Universal Robots PolyScope program: urcadpts_urp_ex.urp

Program urcadpts_urp_ex (installation=default directory=/programs createdIn=5.21.0 lastSavedIn=5.21.0 robotSerialNumber=20205500771)
Calibrated DH parameters: a=[0.00017, -0.315777, -0.390584, 0.000089, 0.000022, 0]; d=[0.16289, -151.810109, 155.986099, -4.043122, 0.099816, 0.099706]; alpha=[1.572969, -0.001875, 0.009547, 1.571313, -1.570827, 0]; deltaTheta=[0, 0.733614, -0.631905, -0.101721, 0.000001, 0]
InitVariablesNode
Robot Program (runOnlyOnce=false)
  Folder Folder
    Folder BeforeStart setup urcadpts: load source file, set PCS and orientation
      'use a script node to load the .script file here'
      Script: urcadpts_set_pcs()
      Script: urcadpts_use_pcs_as_orientation( True )
    Folder RobotProgram Example Usage
      Loop While (checkContinuously=false) expression=urcadpts_pts_remaining()≟ True
        target_point := urcadpts_get_next_point()
        approach_point := pose_trans(target_point, p[0,0,-0.015,0,0,0])
        MoveL speed 50 mm/s, acceleration 100 mm/s^2 (useActiveTCP=true optimoveEnabled=false optiMoveSpeed=0.3 optiMoveAcceleration=0.09) feature=Base
          Waypoint Variable (Variable): variable=approach_point
          Waypoint Variable (Variable): variable=target_point
          Folder Do something when at the target point
            Wait Sleep waitTime=0.5
          Waypoint Variable (Variable): variable=approach_point
